PROGRAM GROUP_1
VAR
	iSetGroupNumber : INT := 1; //SET THIS TO THE NUMBER FOR THIS GROUP
END_VAR

IF _TaskInfo[fbGetCurTaskIndex.index].FirstCycle THEN
	GVL.iAxesGroupIndex := 1;
	FOR GVL.iAxis := 1 TO GVL_APP.nAXIS_NUM DO
		IF astAxes[GVL.iAxis].stDescription.iGroupNumber = iSetGroupNumber THEN
			GVL.astAxesGroup[iSetGroupNumber].aAxesInGroup[GVL.iAxesGroupIndex] := UINT_TO_INT(GVL.iAxis);
			GVL.iAxesGroupIndex := GVL.iAxesGroupIndex + 1;
		END_IF
	END_FOR
	GVL.astAxesGroup[iSetGroupNumber].stDescription.iAxesInGroup := GVL.iAxesGroupIndex -1;
END_IF

END_PROGRAM

(* stored: Version 1.1.0.1, ProductVersion 3.1.4026.18
   POU GROUP_1: Id {941a9b36-9bd6-4e4e-9810-b110625d1266}, SpecialFunc None *)
